{attribute 'Tc2GvlVarNames'}
(* Generated automatically by TwinCAT - do not edit manually! *)
VAR_GLOBAL
END_VAR

(* stored: Version 1.1.0.1, ProductVersion 3.1.4024.15
   GVL TwinCAT_Import: Id {06489816-2cf0-4c99-bb22-754dfc366164} *)
